FUNCTION_BLOCK CiA_DS402Statusword_Danfoss EXTENDS CiA_DS402Statusword
VAR_INPUT
END_VAR
VAR_OUTPUT	
	TargetReached				: BOOL; // Bit 10 in Velocity
	Running						: BOOL; //Bit 14
END_VAR

METHOD PUBLIC readStatusword : BOOL
VAR_INPUT
	Statusword 					:	UINT;
END_VAR


	TargetReached											:= Statusword.10;
	Running													:= Statusword.14;

	readStatusword											:= SUPER^.readStatusword(Statusword);
END_METHOD

END_FUNCTION_BLOCK

(* stored: Version 1.1.0.1, ProductVersion 3.1.4024.3
   POU CiA_DS402Statusword_Danfoss: Id {d2ca5e88-4da8-4963-9294-31309809a690}, SpecialFunc None
   Method readStatusword: Id {05f62b00-e801-43b2-8257-843c71a4a64d} *)
